Staubli VAL3: loadMarkData.pgx

public program loadMarkData(string x_sName, string& x_sMarkList[])
  local num i
  local num j
  local num l_nIndex
  local num l_nSize
  local point l_pPoint
  local string l_sEvent
  local tool l_tTool
begin
  // x_sMarkList

  for i=0 to size(x_sMarkList)-1
    if left(x_sMarkList[i],4)=="TRAJ"
      l_sEvent=right(x_sMarkList[i],len(x_sMarkList[i])-5)
      if isDefined(trajPt:tTraj[l_sEvent])
        // use the type...
        tTraies=trajPt:tTraj[l_sEvent]
      endIf
      l_nSize=size(tTraies.tData)
      for j=0 to l_nSize-1
        if l_nIndex!=0
          insert(sml:box[x_sName].pPointRx[size(sml:box[x_sName].pPointRx)])
          insert(sml:box[x_sName].comment[size(sml:box[x_sName].comment)])
        endIf
        l_pPoint=trajPt:tTraj[l_sEvent].tData[j].pPoint
        pPointRx.trsf=position(l_pPoint,world)
        link(sml:box[x_sName].pPointRx[l_nIndex],world)
        sml:box[x_sName].pPointRx[l_nIndex].trsf=pPointRx.trsf
        sml:box[x_sName].pPointRx[l_nIndex].config=l_pPoint.config
        sml:box[x_sName].comment[l_nIndex]=trajPt:tTraj[l_sEvent].tData[j].tSuper.comment
        l_nIndex=l_nIndex+1
      endFor
      if  sml:box[x_sName].nIndexGun!=tTraies.nIndexTool
        sml:box[x_sName].nIndexGun=tTraies.nIndexTool
      endIf
    endIf
    if left(x_sMarkList[i],6)=="JPOINT"
      l_sEvent=right(x_sMarkList[i],len(x_sMarkList[i])-7)
      if isDefined(jPt:tTraj[l_sEvent])
        // use the type...
        tTrajJoint=jPt:tTraj[l_sEvent]
      endIf
      l_nSize=size(tTrajJoint.tData)
      for j=0 to l_nSize-1
        if l_nIndex!=0
          insert(sml:box[x_sName].pPointRx[size(sml:box[x_sName].pPointRx)])
          insert(sml:box[x_sName].comment[size(sml:box[x_sName].comment)])
        endIf
        l_pPoint=jointToPoint(tTool,world,jPt:tTraj[l_sEvent].tData[j].jJoint)
        link(sml:box[x_sName].pPointRx[l_nIndex],world)
        sml:box[x_sName].pPointRx[l_nIndex].trsf=l_pPoint.trsf
        sml:box[x_sName].pPointRx[l_nIndex].config=l_pPoint.config
        sml:box[x_sName].comment[l_nIndex]=jPt:tTraj[l_sEvent].tData[j].tSuper.comment
        l_nIndex=l_nIndex+1
      endFor
      if  sml:box[x_sName].nIndexGun!=tTrajJoint.nIndexTool
        sml:box[x_sName].nIndexGun=tTrajJoint.nIndexTool
      endIf
    endIf
  endFor

end
